// TIA Portal V16 export
// export: Created 2024-09-05T17:39:21.9047329Z, ExportSetting WithDefaults, DisplayName Totally Integrated Automation Portal, DisplayVersion V16 Update 6, DisplayName TIA Portal Version Control Interface, DisplayVersion V16 Update 2, DisplayName TIA Portal Openness, DisplayVersion V16 Update 6, DisplayName STEP 7 Professional, DisplayVersion V16 Update 6, DisplayName STEP 7 Safety, DisplayVersion V16, DisplayName WinCC Advanced, DisplayVersion V16 Update 6
FUNCTION_BLOCK "Main_Safety_RTG1"   // FB0, F_LAD
{ S7_Optimized_Access := 'TRUE' }
VERSION : 0.1
// stored: AutoNumber false, IsIECCheckEnabled false, UDAEnableTagReadback false
   VAR
      ACK_GL_Instance : ACK_GL;
      "ESTOP1_3L+" : ESTOP1;
      "FDBACK_A2.7" : FDBACK;
      "ESTOP1_4L+" : ESTOP1;
      "FDBACK_A2.8" : FDBACK;
      "FDBACK_A2.9" : FDBACK;
      "ESTOP1_5L+" : ESTOP1;
      "F_IEC_Timer_3L+" : TON;
      "F_IEC_Timer_4L+" : TON;
      FDBACK_KF101x : FDBACK;
      FDBACK_KM20_KM21 : FDBACK;
   END_VAR
BEGIN

REGION Network 1: ACK_GL
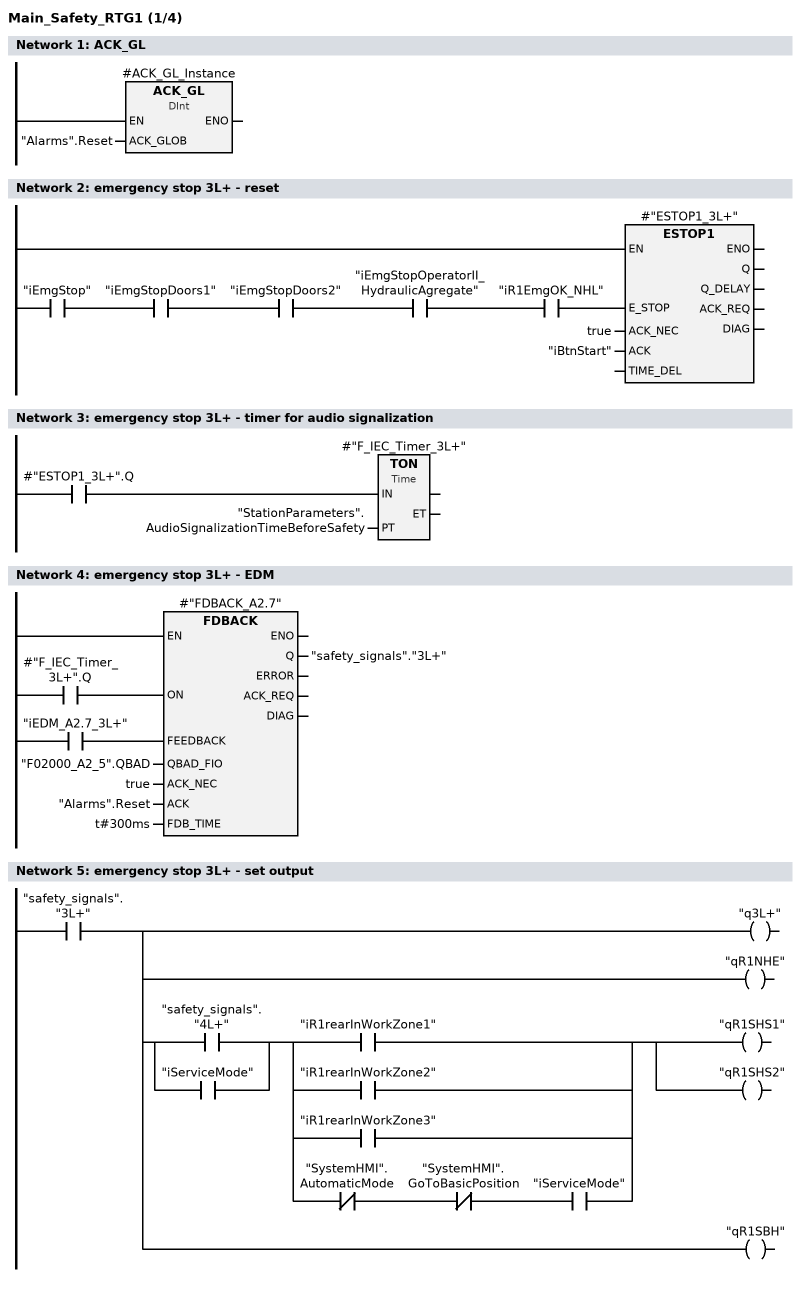
   RUNG wire#powerrail
      { S7_Templates := "codedbool_type := DInt" } #ACK_GL_Instance.ACK_GL(ACK_GLOB := "Alarms".Reset)
   END_RUNG
   // the same network as SCL:
   #ACK_GL_Instance(ACK_GLOB := "Alarms".Reset);   // ACK_GL
END_REGION

REGION Network 2: emergency stop 3L+ - reset
   RUNG wire#powerrail
      #"ESTOP1_3L+".ESTOP1(E_STOP := wire#w1, ACK_NEC := true, ACK := "iBtnStart", TIME_DEL :=, Q =>, Q_DELAY =>, ACK_REQ =>, DIAG =>)
   END_RUNG
   RUNG wire#powerrail
      Contact( "iEmgStop" )
      Contact( "iEmgStopDoors1" )
      Contact( "iEmgStopDoors2" )
      Contact( "iEmgStopOperatorII_HydraulicAgregate" )
      Contact( "iR1EmgOK_NHL" )
   END_RUNG wire#w1
   // the same network as SCL:
   #"ESTOP1_3L+"(E_STOP := "iEmgStop" AND "iEmgStopDoors1" AND "iEmgStopDoors2" AND "iEmgStopOperatorII_HydraulicAgregate" AND "iR1EmgOK_NHL",   // ESTOP1
                 ACK_NEC := true,
                 ACK := "iBtnStart");
END_REGION

REGION Network 3: emergency stop 3L+ - timer for audio signalization
   RUNG wire#powerrail
      Contact( #"ESTOP1_3L+".Q )
      { S7_Templates := "[time_type := Time, codedbool_type := DInt]" } #"F_IEC_Timer_3L+".TON(pt := "StationParameters".AudioSignalizationTimeBeforeSafety, et =>)
   END_RUNG
   // the same network as SCL:
   #"F_IEC_Timer_3L+".TON(IN := #"ESTOP1_3L+".Q, PT := "StationParameters".AudioSignalizationTimeBeforeSafety);
END_REGION

REGION Network 4: emergency stop 3L+ - EDM
   RUNG wire#powerrail
      #"FDBACK_A2.7".FDBACK(ON := wire#w1, FEEDBACK := wire#w2, QBAD_FIO := "F02000_A2_5".QBAD, ACK_NEC := true, ACK := "Alarms".Reset, FDB_TIME := t#300ms, Q => "safety_signals"."3L+", ERROR =>, ACK_REQ =>, DIAG =>)
   END_RUNG
   RUNG wire#powerrail
      Contact( #"F_IEC_Timer_3L+".Q )
   END_RUNG wire#w1
   RUNG wire#powerrail
      Contact( "iEDM_A2.7_3L+" )
   END_RUNG wire#w2
   // the same network as SCL:
   #"FDBACK_A2.7"(ON := #"F_IEC_Timer_3L+".Q,   // FDBACK
                  FEEDBACK := "iEDM_A2.7_3L+",
                  QBAD_FIO := "F02000_A2_5".QBAD,
                  ACK_NEC := true,
                  ACK := "Alarms".Reset,
                  FDB_TIME := t#300ms,
                  Q => "safety_signals"."3L+");
END_REGION

REGION Network 5: emergency stop 3L+ - set output
   RUNG wire#powerrail
      Contact( "safety_signals"."3L+" )
      wire#w1
      Coil( "q3L+" )
   END_RUNG
   RUNG wire#w1
      Coil( "qR1NHE" )
   END_RUNG
   RUNG wire#w1
      Contact( "safety_signals"."4L+" )
      wire#w2
      Contact( "iR1rearInWorkZone1" )
      wire#w3
      Coil( "qR1SHS1" )
   END_RUNG
   RUNG wire#w1
      Contact( "iServiceMode" )
   END_RUNG wire#w2
   RUNG wire#w2
      Contact( "iR1rearInWorkZone2" )
   END_RUNG wire#w3
   RUNG wire#w2
      Contact( "iR1rearInWorkZone3" )
   END_RUNG wire#w3
   RUNG wire#w2
      I_Contact( "SystemHMI".AutomaticMode )
      I_Contact( "SystemHMI".GoToBasicPosition )
      Contact( "iServiceMode" )
   END_RUNG wire#w3
   RUNG wire#w3
      Coil( "qR1SHS2" )
   END_RUNG
   RUNG wire#w1
      Coil( "qR1SBH" )
   END_RUNG
   // the same network as SCL:
   "q3L+" := "safety_signals"."3L+";
   "qR1NHE" := "safety_signals"."3L+";
   "qR1SHS1" := "safety_signals"."3L+" AND ("safety_signals"."4L+" OR "iServiceMode") AND ("iR1rearInWorkZone1" OR "iR1rearInWorkZone2" OR "iR1rearInWorkZone3" OR (NOT "SystemHMI".AutomaticMode AND NOT "SystemHMI".GoToBasicPosition AND "iServiceMode"));
   "qR1SHS2" := "qR1SHS1";
   "qR1SBH" := "safety_signals"."3L+";
END_REGION

REGION Network 6: emergency stop / service doors 4L+ - reset
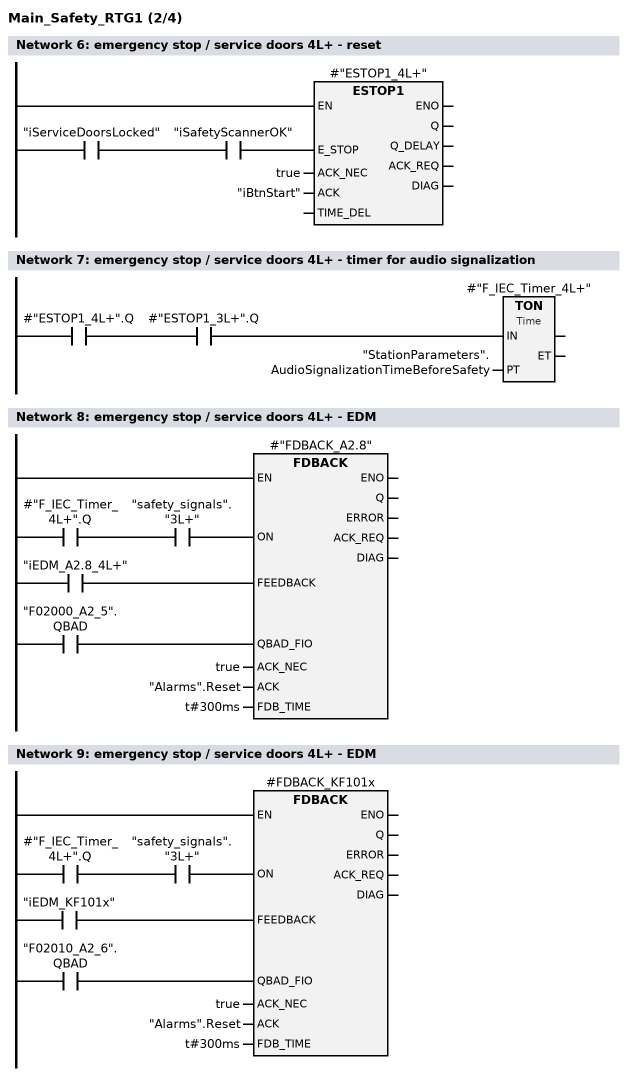
   RUNG wire#powerrail
      #"ESTOP1_4L+".ESTOP1(E_STOP := wire#w1, ACK_NEC := true, ACK := "iBtnStart", TIME_DEL :=, Q =>, Q_DELAY =>, ACK_REQ =>, DIAG =>)
   END_RUNG
   RUNG wire#powerrail
      Contact( "iServiceDoorsLocked" )
      Contact( "iSafetyScannerOK" )
   END_RUNG wire#w1
   // the same network as SCL:
   #"ESTOP1_4L+"(E_STOP := "iServiceDoorsLocked" AND "iSafetyScannerOK", ACK_NEC := true, ACK := "iBtnStart");   // ESTOP1
END_REGION

REGION Network 7: emergency stop / service doors 4L+ - timer for audio signalization
   RUNG wire#powerrail
      Contact( #"ESTOP1_4L+".Q )
      Contact( #"ESTOP1_3L+".Q )
      { S7_Templates := "[time_type := Time, codedbool_type := DInt]" } #"F_IEC_Timer_4L+".TON(pt := "StationParameters".AudioSignalizationTimeBeforeSafety, et =>)
   END_RUNG
   // the same network as SCL:
   #"F_IEC_Timer_4L+".TON(IN := #"ESTOP1_4L+".Q AND #"ESTOP1_3L+".Q,
                          PT := "StationParameters".AudioSignalizationTimeBeforeSafety);
END_REGION

REGION Network 8: emergency stop / service doors 4L+ - EDM
   RUNG wire#powerrail
      #"FDBACK_A2.8".FDBACK(ON := wire#w1, FEEDBACK := wire#w2, QBAD_FIO := wire#w3, ACK_NEC := true, ACK := "Alarms".Reset, FDB_TIME := t#300ms, Q =>, ERROR =>, ACK_REQ =>, DIAG =>)
   END_RUNG
   RUNG wire#powerrail
      Contact( #"F_IEC_Timer_4L+".Q )
      Contact( "safety_signals"."3L+" )
   END_RUNG wire#w1
   RUNG wire#powerrail
      Contact( "iEDM_A2.8_4L+" )
   END_RUNG wire#w2
   RUNG wire#powerrail
      Contact( "F02000_A2_5".QBAD )
   END_RUNG wire#w3
   // the same network as SCL:
   #"FDBACK_A2.8"(ON := #"F_IEC_Timer_4L+".Q AND "safety_signals"."3L+",   // FDBACK
                  FEEDBACK := "iEDM_A2.8_4L+",
                  QBAD_FIO := "F02000_A2_5".QBAD,
                  ACK_NEC := true,
                  ACK := "Alarms".Reset,
                  FDB_TIME := t#300ms);
END_REGION

REGION Network 9: emergency stop / service doors 4L+ - EDM
   RUNG wire#powerrail
      #FDBACK_KF101x.FDBACK(ON := wire#w1, FEEDBACK := wire#w2, QBAD_FIO := wire#w3, ACK_NEC := true, ACK := "Alarms".Reset, FDB_TIME := t#300ms, Q =>, ERROR =>, ACK_REQ =>, DIAG =>)
   END_RUNG
   RUNG wire#powerrail
      Contact( #"F_IEC_Timer_4L+".Q )
      Contact( "safety_signals"."3L+" )
   END_RUNG wire#w1
   RUNG wire#powerrail
      Contact( "iEDM_KF101x" )
   END_RUNG wire#w2
   RUNG wire#powerrail
      Contact( "F02010_A2_6".QBAD )
   END_RUNG wire#w3
   // the same network as SCL:
   #FDBACK_KF101x(ON := #"F_IEC_Timer_4L+".Q AND "safety_signals"."3L+",   // FDBACK
                  FEEDBACK := "iEDM_KF101x",
                  QBAD_FIO := "F02010_A2_6".QBAD,
                  ACK_NEC := true,
                  ACK := "Alarms".Reset,
                  FDB_TIME := t#300ms);
END_REGION

REGION Network 10: emergency stop / service doors 4L+ - set output
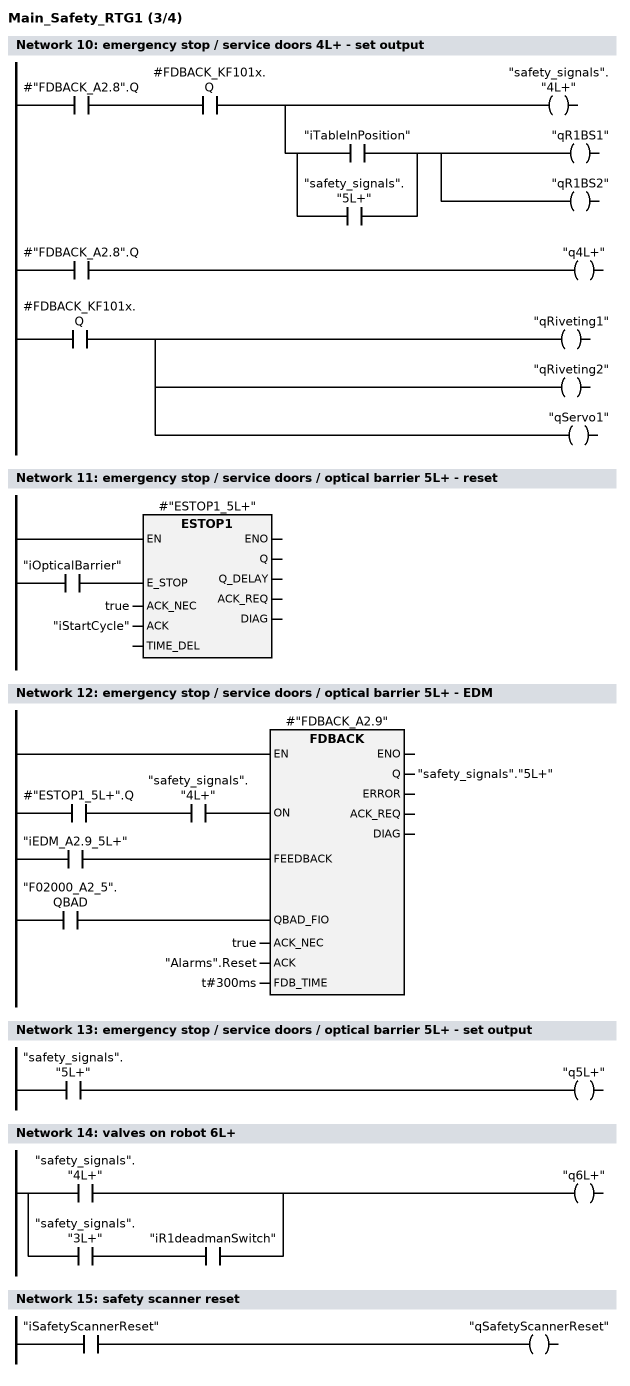
   RUNG wire#powerrail
      Contact( #"FDBACK_A2.8".Q )
      Contact( #FDBACK_KF101x.Q )
      wire#w1
      Coil( "safety_signals"."4L+" )
   END_RUNG
   RUNG wire#w1
      Contact( "iTableInPosition" )
      wire#w2
      Coil( "qR1BS1" )
   END_RUNG
   RUNG wire#w1
      Contact( "safety_signals"."5L+" )
   END_RUNG wire#w2
   RUNG wire#w2
      Coil( "qR1BS2" )
   END_RUNG
   RUNG wire#powerrail
      Contact( #"FDBACK_A2.8".Q )
      Coil( "q4L+" )
   END_RUNG
   RUNG wire#powerrail
      Contact( #FDBACK_KF101x.Q )
      wire#w3
      Coil( "qRiveting1" )
   END_RUNG
   RUNG wire#w3
      Coil( "qRiveting2" )
   END_RUNG
   RUNG wire#w3
      Coil( "qServo1" )
   END_RUNG
   // the same network as SCL:
   "safety_signals"."4L+" := #"FDBACK_A2.8".Q AND #FDBACK_KF101x.Q;
   "qR1BS1" := "safety_signals"."4L+" AND ("iTableInPosition" OR "safety_signals"."5L+");
   "qR1BS2" := "qR1BS1";
   "q4L+" := #"FDBACK_A2.8".Q;
   "qRiveting1" := #FDBACK_KF101x.Q;
   "qRiveting2" := #FDBACK_KF101x.Q;
   "qServo1" := #FDBACK_KF101x.Q;
END_REGION

REGION Network 11: emergency stop / service doors / optical barrier 5L+ - reset
   RUNG wire#powerrail
      #"ESTOP1_5L+".ESTOP1(E_STOP := wire#w1, ACK_NEC := true, ACK := "iStartCycle", TIME_DEL :=, Q =>, Q_DELAY =>, ACK_REQ =>, DIAG =>)
   END_RUNG
   RUNG wire#powerrail
      Contact( "iOpticalBarrier" )
   END_RUNG wire#w1
   // the same network as SCL:
   #"ESTOP1_5L+"(E_STOP := "iOpticalBarrier", ACK_NEC := true, ACK := "iStartCycle");   // ESTOP1
END_REGION

REGION Network 12: emergency stop / service doors / optical barrier 5L+ - EDM
   RUNG wire#powerrail
      #"FDBACK_A2.9".FDBACK(ON := wire#w1, FEEDBACK := wire#w2, QBAD_FIO := wire#w3, ACK_NEC := true, ACK := "Alarms".Reset, FDB_TIME := t#300ms, Q => "safety_signals"."5L+", ERROR =>, ACK_REQ =>, DIAG =>)
   END_RUNG
   RUNG wire#powerrail
      Contact( #"ESTOP1_5L+".Q )
      Contact( "safety_signals"."4L+" )
   END_RUNG wire#w1
   RUNG wire#powerrail
      Contact( "iEDM_A2.9_5L+" )
   END_RUNG wire#w2
   RUNG wire#powerrail
      Contact( "F02000_A2_5".QBAD )
   END_RUNG wire#w3
   // the same network as SCL:
   #"FDBACK_A2.9"(ON := #"ESTOP1_5L+".Q AND "safety_signals"."4L+",   // FDBACK
                  FEEDBACK := "iEDM_A2.9_5L+",
                  QBAD_FIO := "F02000_A2_5".QBAD,
                  ACK_NEC := true,
                  ACK := "Alarms".Reset,
                  FDB_TIME := t#300ms,
                  Q => "safety_signals"."5L+");
END_REGION

REGION Network 13: emergency stop / service doors / optical barrier 5L+ - set output
   RUNG wire#powerrail
      Contact( "safety_signals"."5L+" )
      Coil( "q5L+" )
   END_RUNG
   // the same network as SCL:
   "q5L+" := "safety_signals"."5L+";
END_REGION

REGION Network 14: valves on robot 6L+
   RUNG wire#powerrail
      Contact( "safety_signals"."4L+" )
      wire#w1
      Coil( "q6L+" )
   END_RUNG
   RUNG wire#powerrail
      Contact( "safety_signals"."3L+" )
      Contact( "iR1deadmanSwitch" )
   END_RUNG wire#w1
   // the same network as SCL:
   "q6L+" := "safety_signals"."4L+" OR ("safety_signals"."3L+" AND "iR1deadmanSwitch");
END_REGION

REGION Network 15: safety scanner reset
   RUNG wire#powerrail
      Contact( "iSafetyScannerReset" )
      Coil( "qSafetyScannerReset" )
   END_RUNG
   // the same network as SCL:
   "qSafetyScannerReset" := "iSafetyScannerReset";
END_REGION

REGION Network 16: tool selection for robot - mandatory, but not used
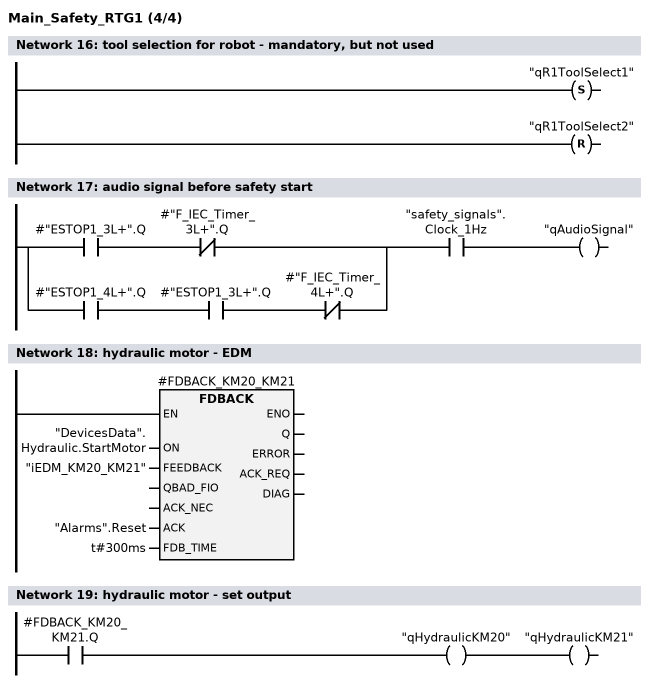
   RUNG wire#powerrail
      S_Coil( "qR1ToolSelect1" )
   END_RUNG
   RUNG wire#powerrail
      R_Coil( "qR1ToolSelect2" )
   END_RUNG
   // the same network as SCL:
   "qR1ToolSelect1" := TRUE;
   "qR1ToolSelect2" := FALSE;
END_REGION

REGION Network 17: audio signal before safety start
   RUNG wire#powerrail
      Contact( #"ESTOP1_3L+".Q )
      I_Contact( #"F_IEC_Timer_3L+".Q )
      wire#w1
      Contact( "safety_signals".Clock_1Hz )
      Coil( "qAudioSignal" )
   END_RUNG
   RUNG wire#powerrail
      Contact( #"ESTOP1_4L+".Q )
      Contact( #"ESTOP1_3L+".Q )
      I_Contact( #"F_IEC_Timer_4L+".Q )
   END_RUNG wire#w1
   // the same network as SCL:
   "qAudioSignal" := ((#"ESTOP1_3L+".Q AND NOT #"F_IEC_Timer_3L+".Q) OR (#"ESTOP1_4L+".Q AND #"ESTOP1_3L+".Q AND NOT #"F_IEC_Timer_4L+".Q)) AND "safety_signals".Clock_1Hz;
END_REGION

REGION Network 18: hydraulic motor - EDM
   RUNG wire#powerrail
      #FDBACK_KM20_KM21.FDBACK(ON := "DevicesData".Hydraulic.StartMotor, FEEDBACK := "iEDM_KM20_KM21", QBAD_FIO :=, ACK_NEC :=, ACK := "Alarms".Reset, FDB_TIME := t#300ms, Q =>, ERROR =>, ACK_REQ =>, DIAG =>)
   END_RUNG
   // the same network as SCL:
   #FDBACK_KM20_KM21(ON := "DevicesData".Hydraulic.StartMotor,   // FDBACK
                     FEEDBACK := "iEDM_KM20_KM21",
                     ACK := "Alarms".Reset,
                     FDB_TIME := t#300ms);
END_REGION

REGION Network 19: hydraulic motor - set output
   RUNG wire#powerrail
      Contact( #FDBACK_KM20_KM21.Q )
      Coil( "qHydraulicKM20" )
      Coil( "qHydraulicKM21" )
   END_RUNG
   // the same network as SCL:
   "qHydraulicKM20" := #FDBACK_KM20_KM21.Q;
   "qHydraulicKM21" := #FDBACK_KM20_KM21.Q;
END_REGION
END_FUNCTION_BLOCK
